FUNCTION_BLOCK PAFVacuum EXTENDS PARoutingFunction
VAR_INPUT
END_VAR
VAR_OUTPUT
END_VAR
VAR
	_ACMethod : ACMethodVacuum;
END_VAR

PROPERTY ACMethod : IACMethod
GET
ACMethod := _ACMethod;
END_GET
END_PROPERTY

METHOD PROTECTED SMIdle
VAR_INPUT
END_VAR
SUPER^.SMIdle();
END_METHOD

METHOD PUBLIC StartWithP : BOOL
VAR_INPUT
	parameter : ACMethodVacuumP;
END_VAR
VAR
	acMethod : ACMethodVacuum;
END_VAR
acMethod.Parameter := parameter;
IF NOT acMethod.IsValid THEN
		StartWithP := FALSE;
	RETURN;
END_IF
_ACMethod.Parameter := parameter;
StartWithP := Start();
END_METHOD

END_FUNCTION_BLOCK

(* stored: Version 1.1.0.1, ProductVersion 3.1.4020.12
   POU PAFVacuum: Id {0e3dbe99-e373-4b59-b22e-d1788ed030c3}, SpecialFunc None
   Folder StateMethods: Id {cd26c9e5-c611-465e-8039-686fb403b360}
   Property ACMethod: Id {d41734cd-4d01-4f1a-a1c2-083f4de9732a}
   Get Get: Id {eb327ea5-5c2f-4c5d-8e86-b85987c58e85}
   Method SMIdle: Id {c9b2db63-53b5-40b2-82dc-e1e7e4f128bd}
   Method StartWithP: Id {648ecb53-1949-469a-a3ab-4b48df1bd9b6} *)
